FUNCTION SUM (* Array Sum *)
  (* Standard: 61499-1 *)
  (* Version 1.0, 2026-01-22, Franz Höpfinger, Andreas Demmler Fahrzeugbau, inspired by SUM in IEC 61131 Paper *)
  PACKAGE logiBUS::utils::dyn_arr;
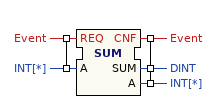
  EVENT_INPUT
    REQ WITH A;
  END_EVENT
  EVENT_OUTPUT
    CNF WITH SUM, A;
  END_EVENT
  VAR_OUTPUT
    SUM : DINT;
  END_VAR
  VAR_IN_OUT
    A : ARRAY [*] OF INT; (* Input *)
  END_VAR
  BODY IN ST:
PACKAGE logiBUS::utils::dyn_arr;

(* Array Sum *)
FUNCTION SUM : DINT

VAR_IN_OUT
	A : ARRAY[*] OF INT; // Input
END_VAR

VAR_TEMP
	i : INT;
	sum2 : DINT;
END_VAR

sum2 := 0;

FOR i := LOWER_BOUND(A,1) TO UPPER_BOUND(A,1) DO
	sum2 := sum2 + A[i];
END_FOR;

SUM := sum2;

END_FUNCTION
  END_BODY
END_FUNCTION
